% RSLogix 500 project lecky_demo.RSS, saved by version 8.30.00.16 %
PROJECT "UNTITLED"    % processor: Bul.1763 MicroLogix 1100 Series B %

PROGRAM FILES
  LAD 2 "CONTINUOUS"  10 rungs
  LAD 252 "2FAILSPLUS"  2 rungs
  LAD 253 "2FAILS5120"  2 rungs
  LAD 254 "2FAILS2560"  2 rungs
  LAD 255 "SYNMPULSES"  6 rungs

DATA FILES
  O0 OUTPUT  4 elements
  I1 INPUT  6 elements
  S2 STATUS  66 elements
  B3 BINARY  1 elements
  T4 TIMER  4 elements
  C5 COUNTER  1 elements
  R6 CONTROL  1 elements
  N7 INTEGER  1 elements
  F8 FLOAT  1 elements
  L9 RJCTTIMERS  1 elements
  B13 MISC_BITS  6 elements
  B103 TMRBSYFLGS  17 elements
  T104 RJCTTIMERS  113 elements

LADDER 2 "CONTINUOUS"
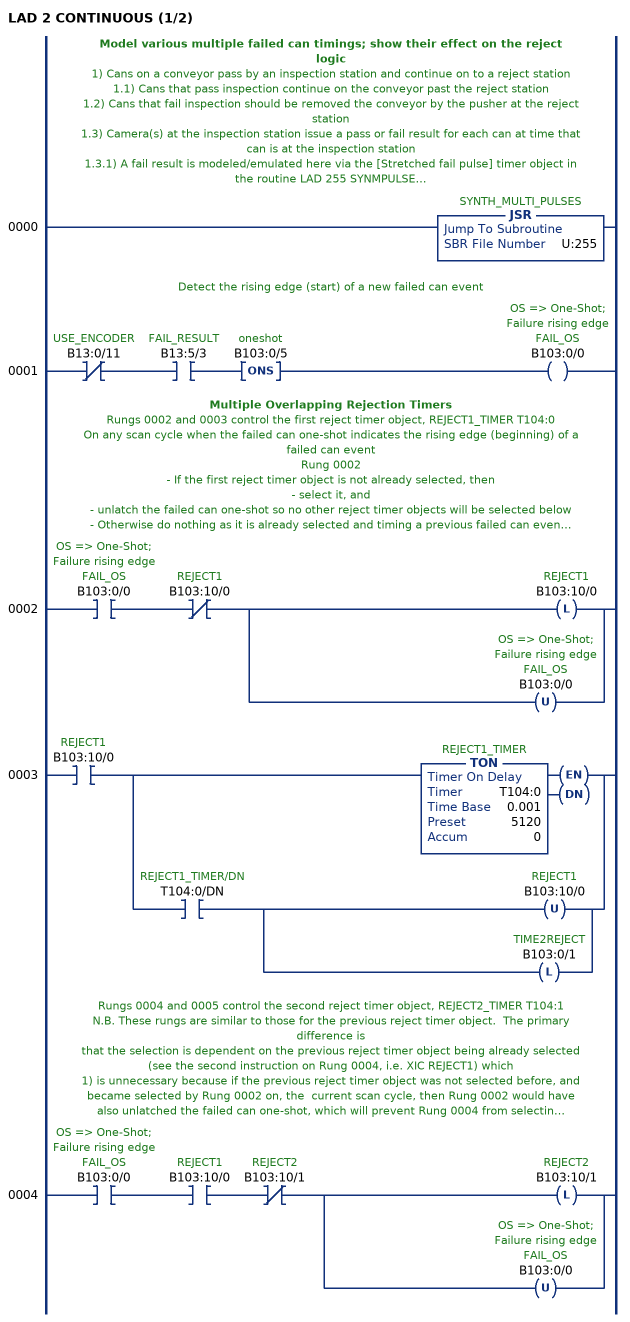
% Rung: 0 %
% TITLE: Model various multiple failed can timings; show their effect on the reject logic %
% 1) Cans on a conveyor pass by an inspection station and continue on to a reject station
% 1.1) Cans that pass inspection continue on the conveyor past the reject station
% 1.2) Cans that fail inspection should be removed the conveyor by the pusher at the reject station
% 1.3) Camera(s) at the inspection station issue a pass or fail result for each can at time that can is at the inspection station
% 1.3.1) A fail result is modeled/emulated here via the [Stretched fail pulse] timer object in the routine LAD 255 SYNMPULSES
% 1.3.2) A pass result is not modeled in this test program program
% 2) On any scan cycle that detects the rising edge of the fail result,
% 2.1) Select the first of the three reject timer objects in Data File T104 that is not already selected by a previous fail event
% 2.1.1) Reject timer object REJECTn_TIMER is not selected when corresponding  bit REJECTn is 0
% 2.1.2) Reject timer object REJECTn_TIMER is selected when corresponding bit REJECTn is 1
% 2.2) Start that reject timer object timing for 5120ms (5.12s) in a TON (Timer ON-delay) instruction
% 3) The reject timer object's increasing accumulation of time models the motion of the failed can
%       from the inspection station,  along the conveyor, to the reject station
% 4) When a reject timer object expires (T104:x/DN bit will be 1),
% 4.1) The failed can, which selected that reject timer object, is assumed, in the model, to be
%          in front of the reject pusher solenoid.
% 4.2) Set the reject bit (TIME2REJECT) to 1 to trigger the solenoid and reject the failed can
% 3.2) Deselect that reject timer object (reset its reject bit to 0)
% ========================================================================
% 
% Rung 0000 calls the routine LAD 255 SYNMPULSES, which emulates particular timings
% of failed cans detected by the camera(s) at the inspection station; refer to the comments in
% routine SYNMPULSES for more detail. %
SOR JSR U:255 EOR
%   U:255  SYNTH_MULTI_PULSES %
% Rung: 1 %
% Detect the rising edge (start) of a new failed can event %
SOR XIO B13:0/11 XIC B13:5/3 ONS B103:0/5 OTE B103:0/0 EOR
%   B13:0/11  USE_ENCODER %
%   B13:5/3  FAIL_RESULT %
%   B103:0/5  "oneshot" %
%   B103:0/0  FAIL_OS  "OS => One-Shot; Failure rising edge" %
% Rung: 2 %
% TITLE: Multiple Overlapping Rejection Timers %
% Rungs 0002 and 0003 control the first reject timer object, REJECT1_TIMER T104:0
% 
% On any scan cycle when the failed can one-shot indicates the rising edge (beginning) of a failed can event
% Rung 0002
%     - If the first reject timer object is not already selected, then
%          - select it, and
%          - unlatch the failed can one-shot so no other reject timer objects will be selected below
%     - Otherwise do nothing as it is already selected and timing a previous failed can event
% Rung 0004
%     - If the first reject timer object has been selected, then start and continue its timing for 5120ms*
%     - When the first timer object expires, deselect it
% 
% * N.B. the timer object preset of 5.12s was chosen to make it easier to observe
%              the behavior of  reject logic in this demonstration program, and is, and
%              is not meant to represent an actual conveyor line. %
SOR XIC B103:0/0 XIO B103:10/0 BST OTL B103:10/0 NXB OTU B103:0/0 BND EOR
%   B103:0/0  FAIL_OS  "OS => One-Shot; Failure rising edge" %
%   B103:10/0  REJECT1 %
% Rung: 3 %
SOR XIC B103:10/0 BST TON T104:0 0.001 5120 0 NXB XIC T104:0/DN BST OTU B103:10/0 NXB OTL B103:0/1 BND BND EOR
%   B103:10/0  REJECT1 %
%   T104:0  REJECT1_TIMER %
%   B103:0/1  TIME2REJECT %
% Rung: 4 %
% Rungs 0004 and 0005 control the second reject timer object, REJECT2_TIMER T104:1
% 
% N.B. These rungs are similar to those for the previous reject timer object.  The primary difference is
%           that the selection is dependent on the previous reject timer object being already selected
%            (see the second instruction on Rung 0004, i.e. XIC REJECT1) which
% 
%             1) is unnecessary because if the previous reject timer object was not selected before, and
%                  became selected by Rung 0002 on, the  current scan cycle, then Rung 0002 would have
%                  also unlatched the failed can one-shot, which will prevent Rung 0004 from selecting
%                  the second timer object for the same failed can,
% 
%              2) is also a design error, because if the first timer object above expired on the current scan
%                   cycle, then the first reject timer object selection bit (REJECT1)
%                   2.1) would have been latched when evaluating Rung 0002, which would prevent the first
%                            timer object from being selected by the current failed can event, and
%                    2.2) would have been unlatched after evaluating Rung 0003, because the first timer
%                             object expired,
%                    2.3) and finally, on this Rung 0004, that unlatched state of  that first reject timer object
%                             selection bit would prevent selection of  the second reject timer object, even
%                             though that second reject timer object was not selected. %
SOR XIC B103:0/0 XIC B103:10/0 XIO B103:10/1 BST OTL B103:10/1 NXB OTU B103:0/0 BND EOR
%   B103:0/0  FAIL_OS  "OS => One-Shot; Failure rising edge" %
%   B103:10/0  REJECT1 %
%   B103:10/1  REJECT2 %

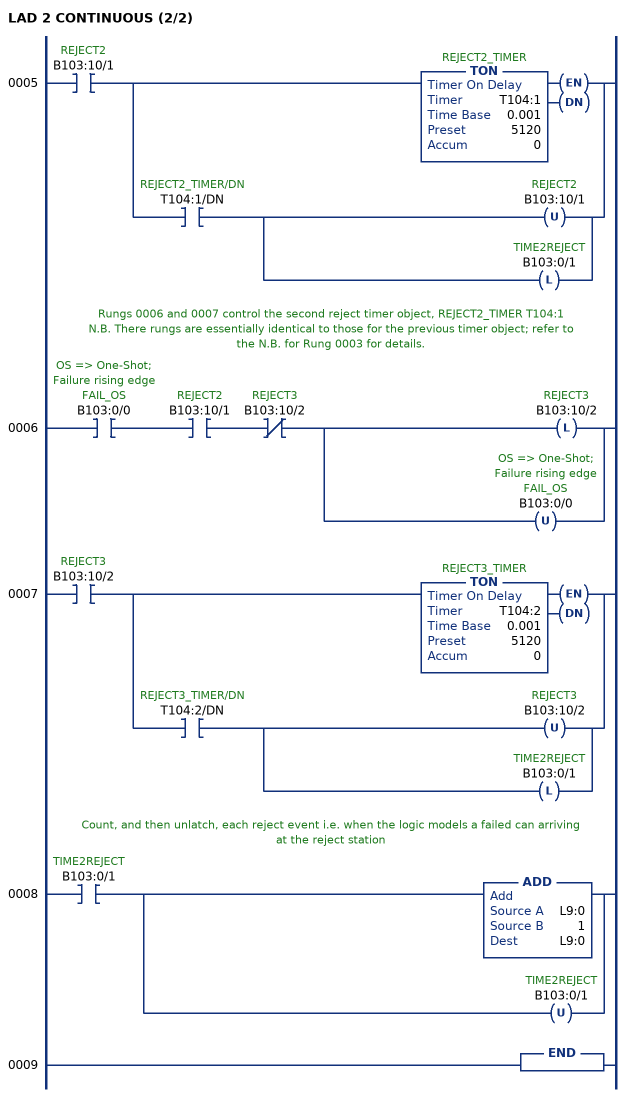
% Rung: 5 %
SOR XIC B103:10/1 BST TON T104:1 0.001 5120 0 NXB XIC T104:1/DN BST OTU B103:10/1 NXB OTL B103:0/1 BND BND EOR
%   B103:10/1  REJECT2 %
%   T104:1  REJECT2_TIMER %
%   B103:0/1  TIME2REJECT %
% Rung: 6 %
% Rungs 0006 and 0007 control the second reject timer object, REJECT2_TIMER T104:1
% 
% N.B. There rungs are essentially identical to those for the previous timer object; refer to
%           the N.B. for Rung 0003 for details. %
SOR XIC B103:0/0 XIC B103:10/1 XIO B103:10/2 BST OTL B103:10/2 NXB OTU B103:0/0 BND EOR
%   B103:0/0  FAIL_OS  "OS => One-Shot; Failure rising edge" %
%   B103:10/1  REJECT2 %
%   B103:10/2  REJECT3 %
% Rung: 7 %
SOR XIC B103:10/2 BST TON T104:2 0.001 5120 0 NXB XIC T104:2/DN BST OTU B103:10/2 NXB OTL B103:0/1 BND BND EOR
%   B103:10/2  REJECT3 %
%   T104:2  REJECT3_TIMER %
%   B103:0/1  TIME2REJECT %
% Rung: 8 %
% Count, and then unlatch, each reject event i.e. when the logic models a failed can arriving at the reject station %
SOR XIC B103:0/1 BST ADD L9:0 1 L9:0 NXB OTU B103:0/1 BND EOR
%   B103:0/1  TIME2REJECT %
% Rung: 9 %
SOR END EOR

LADDER 252 "2FAILSPLUS"
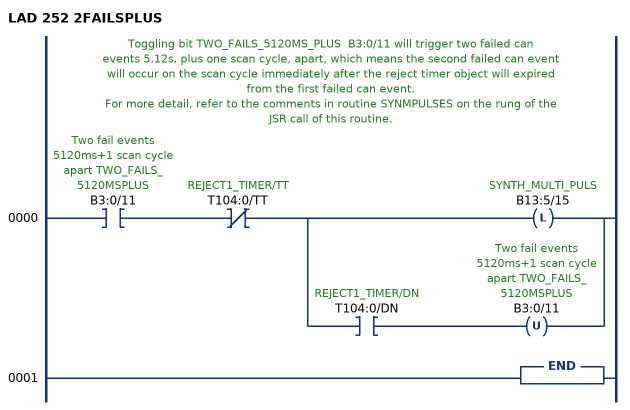
% Rung: 0 %
% Toggling bit TWO_FAILS_5120MS_PLUS  B3:0/11 will trigger two failed can
% events 5.12s, plus one scan cycle, apart, which means the second failed can event
% will occur on the scan cycle immediately after the reject timer object will expired
% from the first failed can event.
% 
% For more detail, refer to the comments in routine SYNMPULSES on the rung of the
% JSR call of this routine. %
SOR XIC B3:0/11 XIO T104:0/TT BST OTL B13:5/15 NXB XIC T104:0/DN OTU B3:0/11 BND EOR
%   B3:0/11  TWO_FAILS_5120MSPLUS  "Two fail events 5120ms+1 scan cycle apart" %
%   T104:0  REJECT1_TIMER %
%   B13:5/15  SYNTH_MULTI_PULS %
% Rung: 1 %
SOR END EOR

LADDER 253 "2FAILS5120"
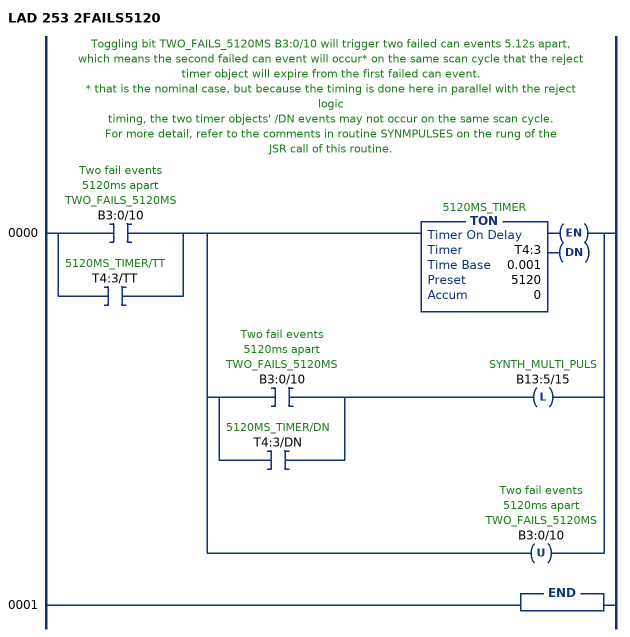
% Rung: 0 %
% Toggling bit TWO_FAILS_5120MS B3:0/10 will trigger two failed can events 5.12s apart,
% which means the second failed can event will occur* on the same scan cycle that the reject
% timer object will expire from the first failed can event.
% 
% * that is the nominal case, but because the timing is done here in parallel with the reject logic
%     timing, the two timer objects' /DN events may not occur on the same scan cycle.
% 
% For more detail, refer to the comments in routine SYNMPULSES on the rung of the
% JSR call of this routine. %
SOR BST XIC B3:0/10 NXB XIC T4:3/TT BND BST TON T4:3 0.001 5120 0 NXB BST XIC B3:0/10 NXB XIC T4:3/DN BND OTL B13:5/15 NXB OTU B3:0/10 BND EOR
%   B3:0/10  TWO_FAILS_5120MS  "Two fail events 5120ms apart" %
%   T4:3  5120MS_TIMER %
%   B13:5/15  SYNTH_MULTI_PULS %
% Rung: 1 %
SOR END EOR

LADDER 254 "2FAILS2560"
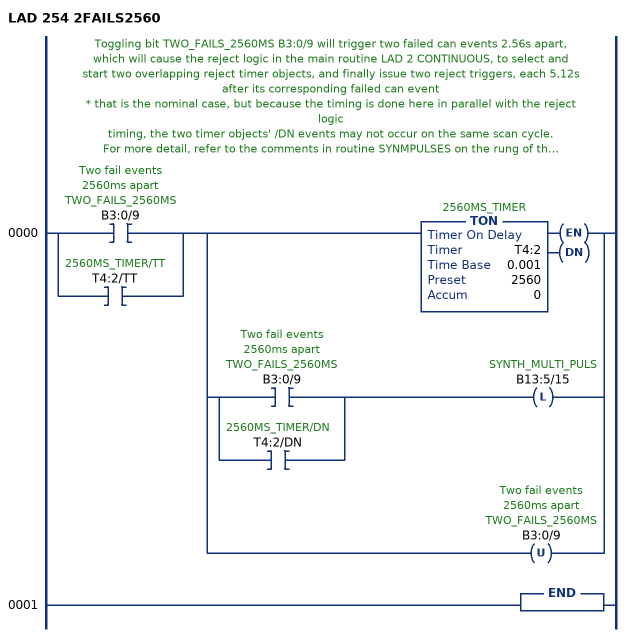
% Rung: 0 %
% Toggling bit TWO_FAILS_2560MS B3:0/9 will trigger two failed can events 2.56s apart,
% which will cause the reject logic in the main routine LAD 2 CONTINUOUS, to select and
% start two overlapping reject timer objects, and finally issue two reject triggers, each 5.12s
% after its corresponding failed can event
% 
% * that is the nominal case, but because the timing is done here in parallel with the reject logic
%     timing, the two timer objects' /DN events may not occur on the same scan cycle.
% 
% For more detail, refer to the comments in routine SYNMPULSES on the rung of the
% JSR call of this routine. %
SOR BST XIC B3:0/9 NXB XIC T4:2/TT BND BST TON T4:2 0.001 2560 0 NXB BST XIC B3:0/9 NXB XIC T4:2/DN BND OTL B13:5/15 NXB OTU B3:0/9 BND EOR
%   B3:0/9  TWO_FAILS_2560MS  "Two fail events 2560ms apart" %
%   T4:2  2560MS_TIMER %
%   B13:5/15  SYNTH_MULTI_PULS %
% Rung: 1 %
SOR END EOR

LADDER 255 "SYNMPULSES"
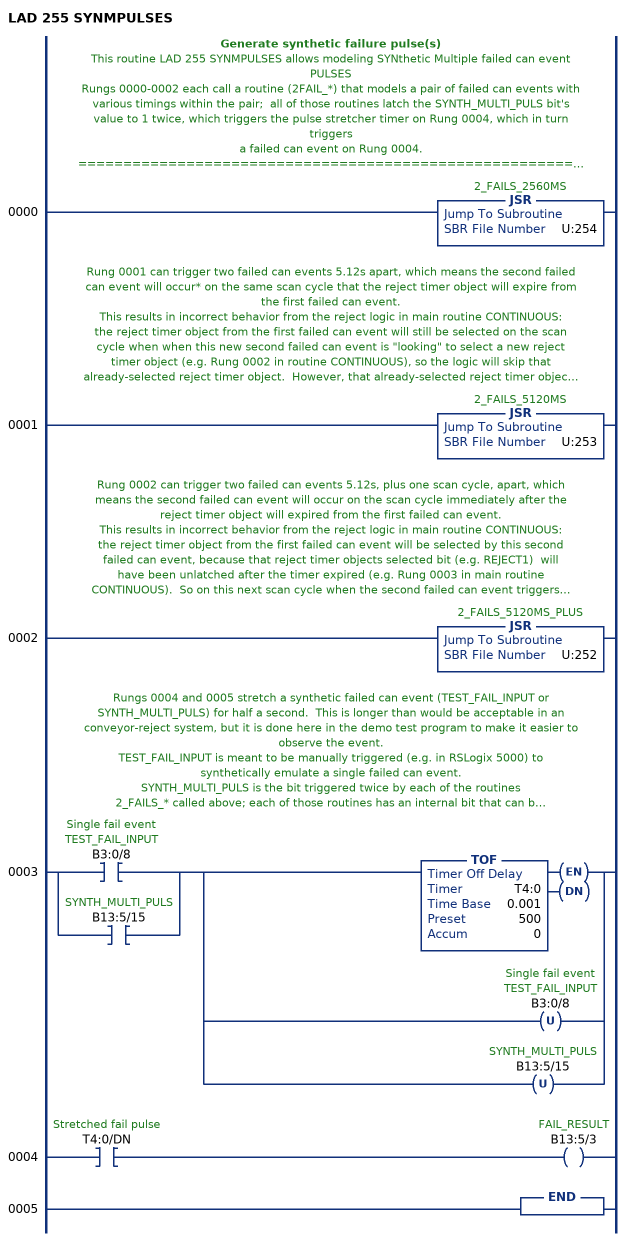
% Rung: 0 %
% TITLE: Generate synthetic failure pulse(s) %
% This routine LAD 255 SYNMPULSES allows modeling SYNthetic Multiple failed can event PULSES
% 
% Rungs 0000-0002 each call a routine (2FAIL_*) that models a pair of failed can events with
% various timings within the pair;  all of those routines latch the SYNTH_MULTI_PULS bit's
% value to 1 twice, which triggers the pulse stretcher timer on Rung 0004, which in turn triggers
% a failed can event on Rung 0004.
% ========================================================================
% 
% Rung 0000 can trigger two failed can events 2.56s apart, which will cause the reject logic in
% the main routine LAD 2 CONTINUOUS, to select and start two overlapping reject timer
% objects, and finally issue two reject triggers, each 5.12s after its corresponding failed can event
% 
% This triggers correct behavior from the reject logic in main routine CONTINUOUS %
SOR JSR U:254 EOR
%   U:254  2_FAILS_2560MS %
% Rung: 1 %
% Rung 0001 can trigger two failed can events 5.12s apart, which means the second failed
% can event will occur* on the same scan cycle that the reject timer object will expire from
% the first failed can event.
% 
% This results in incorrect behavior from the reject logic in main routine CONTINUOUS:
% the reject timer object from the first failed can event will still be selected on the scan
% cycle when when this new second failed can event is "looking" to select a new reject
% timer object (e.g. Rung 0002 in routine CONTINUOUS), so the logic will skip that
% already-selected reject timer object.  However, that already-selected reject timer object
% will also expire on the next rung on that same scan cycle, which expiry will unlatch
% the selected bit (e.g. Rung 0003 in routine CONTINUOUS; bit REJECT1), and that
% unlatched bit will prevent the next reject timer object from being selected on the
% following rung (e.g. Rung 0004 in routine CONTINOUUS; see the instruction
% XIC REJECT1).
% 
% * that is the nominal case, but because the timing is done here in parallel with the reject logic
%     timing, the two timer objects' /DN events may not occur on the same scan cycle. %
SOR JSR U:253 EOR
%   U:253  2_FAILS_5120MS %
% Rung: 2 %
% Rung 0002 can trigger two failed can events 5.12s, plus one scan cycle, apart, which
% means the second failed can event will occur on the scan cycle immediately after the
% reject timer object will expired from the first failed can event.
% 
% This results in incorrect behavior from the reject logic in main routine CONTINUOUS:
% the reject timer object from the first failed can event will be selected by this second
% failed can event, because that reject timer objects selected bit (e.g. REJECT1)  will
% have been unlatched after the timer expired (e.g. Rung 0003 in main routine
% CONTINUOUS).  So on this next scan cycle when the second failed can event triggers,
% the feed rung into the TON instruction will be true, and since it was also true on the
% previous scan cycle i.e. when it expired from the first failed can event, the reject timer
% object will still be enabled as well as expired, so it will immediately issue a second
% reject trigger by latching the value of TIMER2REJECT to 1 (e.g. Rung 0003 in main
% routine CONTINUOUS).. %
SOR JSR U:252 EOR
%   U:252  2_FAILS_5120MS_PLUS %
% Rung: 3 %
% Rungs 0004 and 0005 stretch a synthetic failed can event (TEST_FAIL_INPUT or
% SYNTH_MULTI_PULS) for half a second.  This is longer than would be acceptable in an
% conveyor-reject system, but it is done here in the demo test program to make it easier to
% observe the event.
% 
% TEST_FAIL_INPUT is meant to be manually triggered (e.g. in RSLogix 5000) to
% synthetically emulate a single failed can event.
% 
% SYNTH_MULTI_PULS is the bit triggered twice by each of the routines
% 2_FAILS_* called above; each of those routines has an internal bit that can be
% triggered manually to trigger the two latches of SYNTH_MULTI_PULS at the
% timing apropos whichever 2_FAILS_* internal bit is manually triggered. %
SOR BST XIC B3:0/8 NXB XIC B13:5/15 BND BST TOF T4:0 0.001 500 0 NXB OTU B3:0/8 NXB OTU B13:5/15 BND EOR
%   B3:0/8  TEST_FAIL_INPUT  "Single fail event" %
%   B13:5/15  SYNTH_MULTI_PULS %
% Rung: 4 %
SOR XIC T4:0/DN OTE B13:5/3 EOR
%   T4:0/DN  "Stretched fail pulse" %
%   B13:5/3  FAIL_RESULT %
% Rung: 5 %
SOR END EOR

DATA TABLE (non-zero values as saved)
DATA T4
% .PRE .ACC %
% T4:0 % 500 0
% T4:1 % 51 0
% T4:2 % 2560 0
% T4:3 % 5120 0
DATA C5
% .PRE .ACC %
% C5:0 % 6001 0
DATA T104
% .PRE .ACC %
% T104:0 % 5120 0
% T104:1 % 5120 0
% T104:2 % 5120 0
